PROGRAM p_Com_Modbus_RS485
VAR
	//Gestion de la com avec la passerelle LED
	Com_LED: Com485_Dalcnet;
	Lecture_Dimmer 	:INT;
	Lecture_Rouge 	:INT;
	Lecture_Vert 	:INT;
	Lecture_Bleu 	:INT;
	Lecture_Blanc 	:INT;
	LED_Com_Ok		:BOOL;
	LED_Com_Error	:BOOL;
	LED_Etape		:INT;
	
	//Gestion de la com avec GVL_RegTROX.Reg_Souf_GD_FCVT01
	FCVT01_Com_Ok		:BOOL;
	FCVT01_Com_Error	:BOOL;
	FCVT01_Etape		:INT;
	FCVT01_ConsAppli	:INT;
	
	//Gestion de la com avec GVL_RegTROX.Com_RegSouf_PD_FCVT02
	FCVT02_Com_Ok		:BOOL;
	FCVT02_Com_Error	:BOOL;
	FCVT02_Etape		:INT;
	FCVT02_ConsAppli	:INT;
	
	//Gestion de la com avec GVL_RegTROX.Com_RegSouf_Cabine_FCVT03
	FCVT03_Com_Ok		:BOOL;
	FCVT03_Com_Error	:BOOL;
	FCVT03_Etape		:INT;
	FCVT03_ConsAppli	:INT;
	
	//Gestion de la com avec GVL_RegTROX.Com_Reg_Bypass_FCVT04
	FCVT04_Com_Ok		:BOOL;
	FCVT04_Com_Error	:BOOL;
	FCVT04_Etape		:INT;
	FCVT04_ConsAppli	:INT;
	
	//Gestion de la com avec GVL_RegTROX.Com_RegSouf_CabGD_FCVT05
	FCVT05_Com_Ok		:BOOL;
	FCVT05_Com_Error	:BOOL;
	FCVT05_Etape		:INT;
	FCVT05_ConsAppli	:INT;
	
	//Gestion de la com avec GVL_RegTROX.Com_RegSouf_CabPD_FCVT06
	FCVT06_Com_Ok		:BOOL;
	FCVT06_Com_Error	:BOOL;
	FCVT06_Etape		:INT;
	FCVT06_ConsAppli	:INT;
	
	//Gestion de la com avec GVL_RegTROX.Com_RegRep_FCVT07
	FCVT07_Com_Ok		:BOOL;
	FCVT07_Com_Error	:BOOL;
	FCVT07_Etape		:INT;
	FCVT07_ConsAppli	:INT;
	
	Start_2: BOOL;
	Start_3: BOOL;
	Start_4: BOOL;
	Start_41: BOOL;
	Start_5: BOOL;
	Start_6: BOOL;
	Start_61: BOOL;
	Start_7: BOOL;
	Start_8: BOOL;
	Start_9: BOOL;
	FirstCycle: BOOL := TRUE;
	F_TRIG_0: F_TRIG;
	cpt: INT;
	CTU_Cpt: CTU;
	Cons_Cpt: WORD := 4;
	TOF_0: TOF;
	test: BOOL;
	
	//Gestion des forçages
	EF_FCVT01		:BOOL;
	F_FCVT01		:REAL;
	EF_FCVT02		:BOOL;
	F_FCVT02		:REAL;
	EF_FCVT03		:BOOL;
	F_FCVT03		:REAL;
	EF_FCVT04		:BOOL;
	F_FCVT04		:REAL;
	EF_FCVT05		:BOOL;
	F_FCVT05		:REAL;
	EF_FCVT06		:BOOL;
	F_FCVT06		:REAL;
	EF_FCVT07		:BOOL;
	F_FCVT07		:REAL;
END_VAR
VAR // added by the converter: edge detectors and wires of the graphical bodies
    _w1 : BOOL;
END_VAR

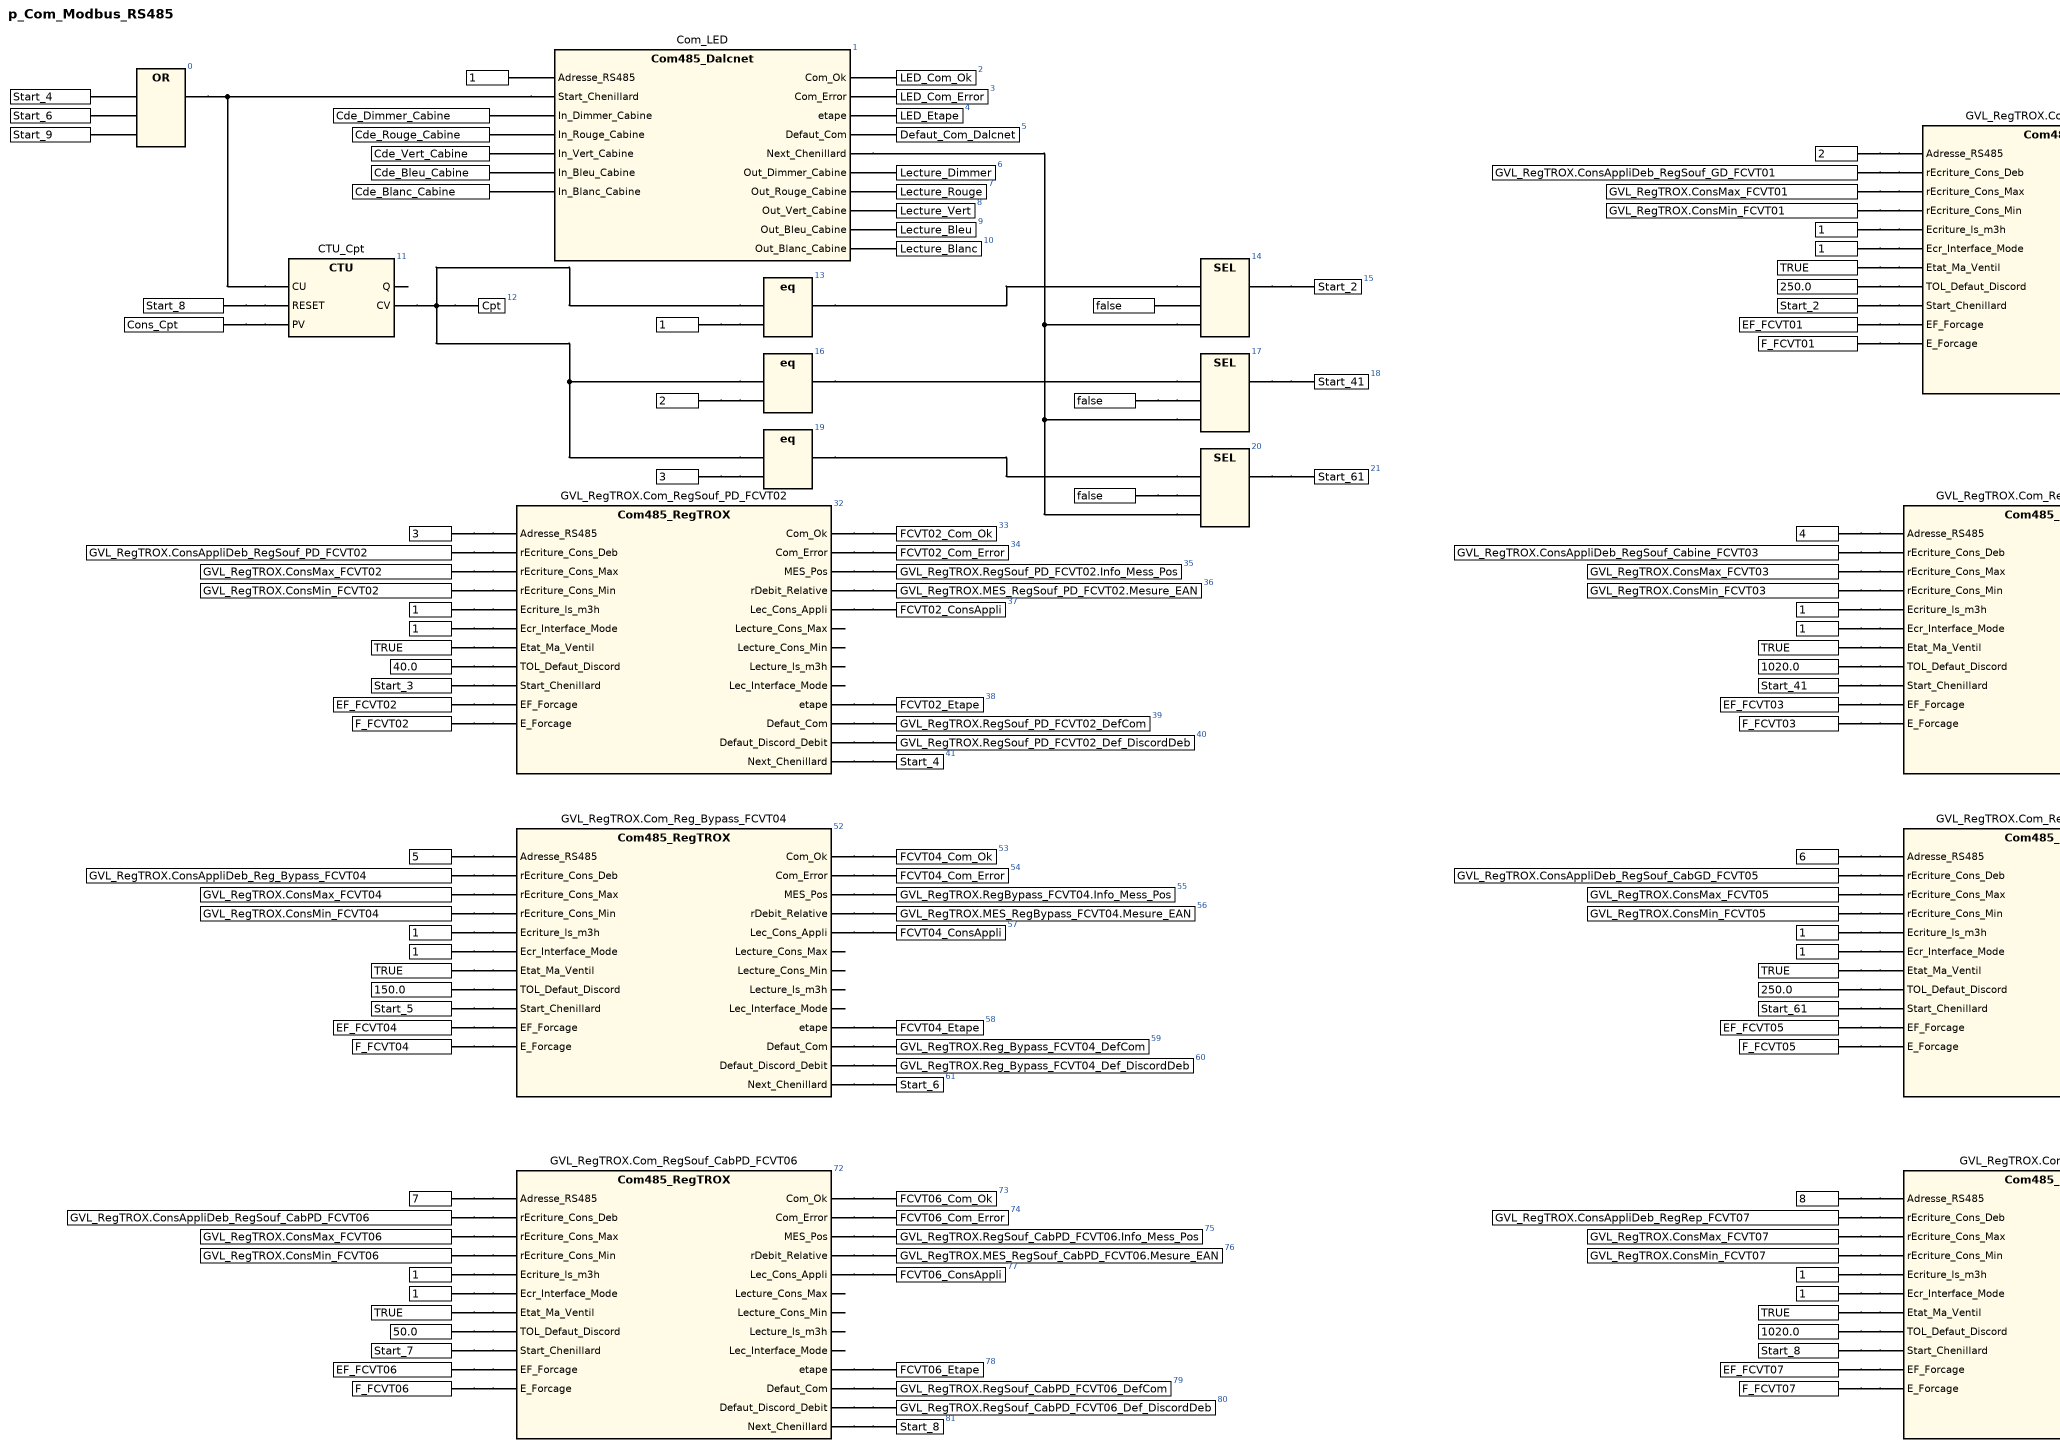
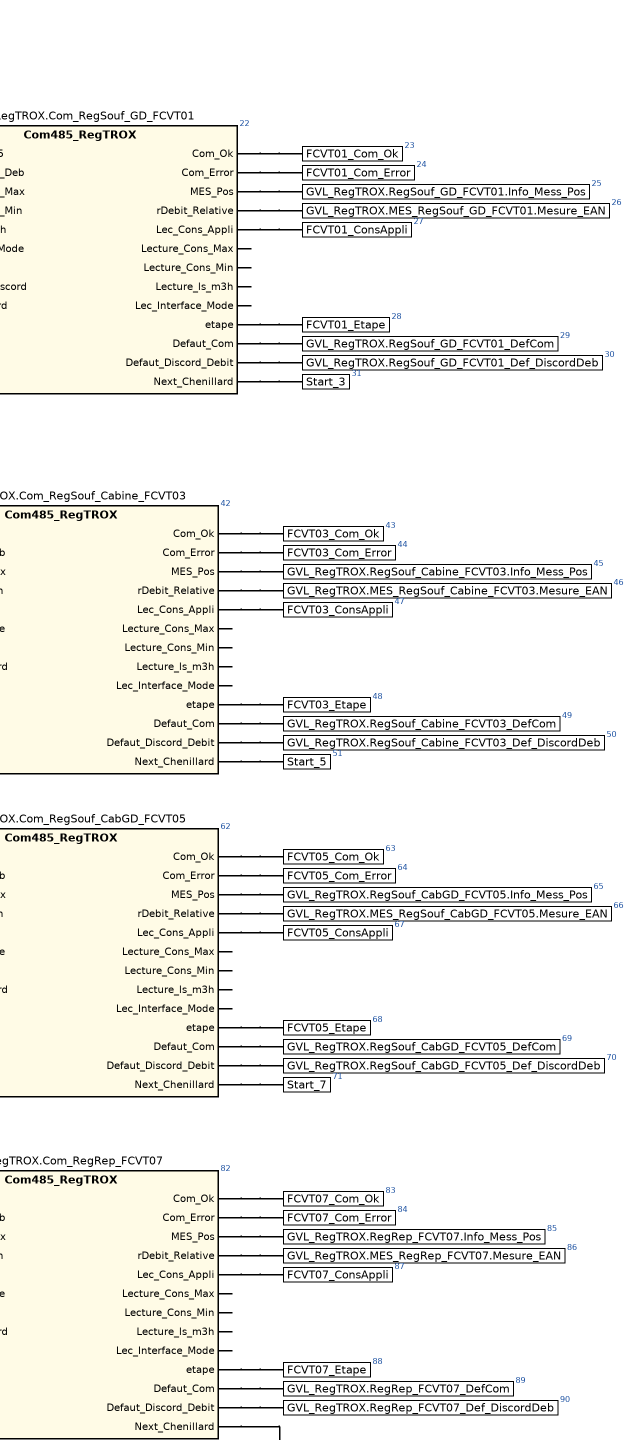
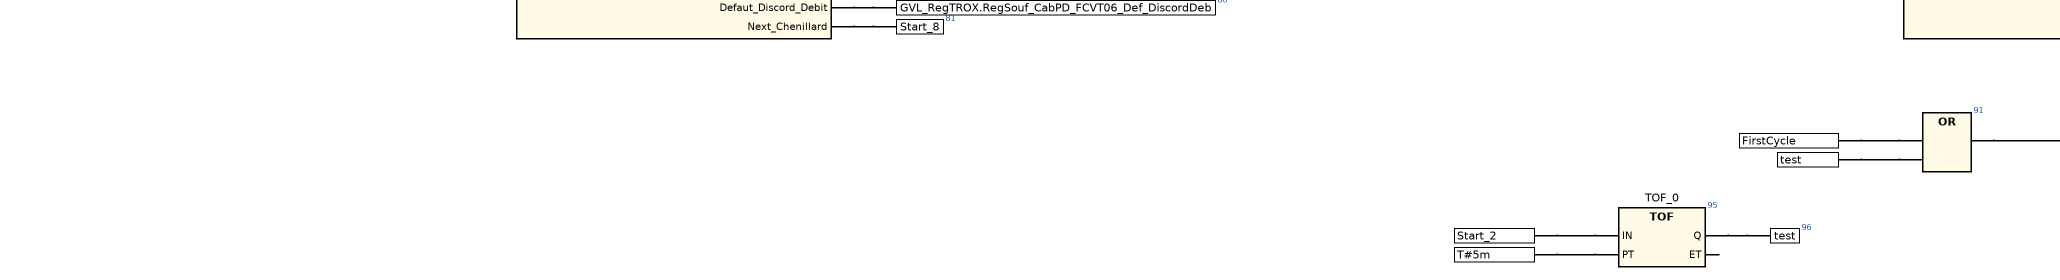
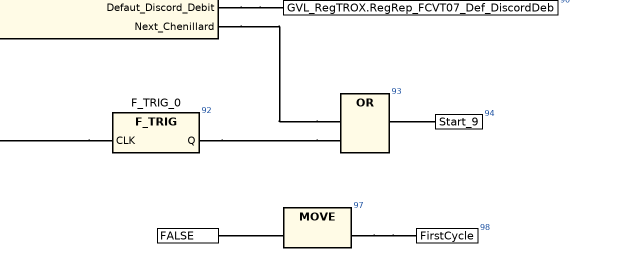
_w1 := Start_4 OR Start_6 OR Start_9;
Com_LED(
    Adresse_RS485 := 1,
    Start_Chenillard := _w1,
    In_Dimmer_Cabine := Cde_Dimmer_Cabine,
    In_Rouge_Cabine := Cde_Rouge_Cabine,
    In_Vert_Cabine := Cde_Vert_Cabine,
    In_Bleu_Cabine := Cde_Bleu_Cabine,
    In_Blanc_Cabine := Cde_Blanc_Cabine); // Com485_Dalcnet
LED_Com_Ok := Com_LED.Com_Ok;
LED_Com_Error := Com_LED.Com_Error;
LED_Etape := Com_LED.etape;
Defaut_Com_Dalcnet := Com_LED.Defaut_Com;
Lecture_Dimmer := Com_LED.Out_Dimmer_Cabine;
Lecture_Rouge := Com_LED.Out_Rouge_Cabine;
Lecture_Vert := Com_LED.Out_Vert_Cabine;
Lecture_Bleu := Com_LED.Out_Bleu_Cabine;
Lecture_Blanc := Com_LED.Out_Blanc_Cabine;
CTU_Cpt(CU := _w1, RESET := Start_8, PV := Cons_Cpt); // CTU
Cpt := CTU_Cpt.CV;
Start_2 := SEL(CTU_Cpt.CV = 1, false, Com_LED.Next_Chenillard);
Start_41 := SEL(CTU_Cpt.CV = 2, false, Com_LED.Next_Chenillard);
Start_61 := SEL(CTU_Cpt.CV = 3, false, Com_LED.Next_Chenillard);
GVL_RegTROX.Com_RegSouf_GD_FCVT01(
    Adresse_RS485 := 2,
    rEcriture_Cons_Deb := GVL_RegTROX.ConsAppliDeb_RegSouf_GD_FCVT01,
    rEcriture_Cons_Max := GVL_RegTROX.ConsMax_FCVT01,
    rEcriture_Cons_Min := GVL_RegTROX.ConsMin_FCVT01,
    Ecriture_ls_m3h := 1,
    Ecr_Interface_Mode := 1,
    Etat_Ma_Ventil := TRUE,
    TOL_Defaut_Discord := 250.0,
    Start_Chenillard := Start_2,
    EF_Forcage := EF_FCVT01,
    E_Forcage := F_FCVT01); // Com485_RegTROX
FCVT01_Com_Ok := GVL_RegTROX.Com_RegSouf_GD_FCVT01.Com_Ok;
FCVT01_Com_Error := GVL_RegTROX.Com_RegSouf_GD_FCVT01.Com_Error;
GVL_RegTROX.RegSouf_GD_FCVT01.Info_Mess_Pos := GVL_RegTROX.Com_RegSouf_GD_FCVT01.MES_Pos;
GVL_RegTROX.MES_RegSouf_GD_FCVT01.Mesure_EAN := GVL_RegTROX.Com_RegSouf_GD_FCVT01.rDebit_Relative;
FCVT01_ConsAppli := GVL_RegTROX.Com_RegSouf_GD_FCVT01.Lec_Cons_Appli;
FCVT01_Etape := GVL_RegTROX.Com_RegSouf_GD_FCVT01.etape;
GVL_RegTROX.RegSouf_GD_FCVT01_DefCom := GVL_RegTROX.Com_RegSouf_GD_FCVT01.Defaut_Com;
GVL_RegTROX.RegSouf_GD_FCVT01_Def_DiscordDeb := GVL_RegTROX.Com_RegSouf_GD_FCVT01.Defaut_Discord_Debit;
Start_3 := GVL_RegTROX.Com_RegSouf_GD_FCVT01.Next_Chenillard;
GVL_RegTROX.Com_RegSouf_PD_FCVT02(
    Adresse_RS485 := 3,
    rEcriture_Cons_Deb := GVL_RegTROX.ConsAppliDeb_RegSouf_PD_FCVT02,
    rEcriture_Cons_Max := GVL_RegTROX.ConsMax_FCVT02,
    rEcriture_Cons_Min := GVL_RegTROX.ConsMin_FCVT02,
    Ecriture_ls_m3h := 1,
    Ecr_Interface_Mode := 1,
    Etat_Ma_Ventil := TRUE,
    TOL_Defaut_Discord := 40.0,
    Start_Chenillard := Start_3,
    EF_Forcage := EF_FCVT02,
    E_Forcage := F_FCVT02); // Com485_RegTROX
FCVT02_Com_Ok := GVL_RegTROX.Com_RegSouf_PD_FCVT02.Com_Ok;
FCVT02_Com_Error := GVL_RegTROX.Com_RegSouf_PD_FCVT02.Com_Error;
GVL_RegTROX.RegSouf_PD_FCVT02.Info_Mess_Pos := GVL_RegTROX.Com_RegSouf_PD_FCVT02.MES_Pos;
GVL_RegTROX.MES_RegSouf_PD_FCVT02.Mesure_EAN := GVL_RegTROX.Com_RegSouf_PD_FCVT02.rDebit_Relative;
FCVT02_ConsAppli := GVL_RegTROX.Com_RegSouf_PD_FCVT02.Lec_Cons_Appli;
FCVT02_Etape := GVL_RegTROX.Com_RegSouf_PD_FCVT02.etape;
GVL_RegTROX.RegSouf_PD_FCVT02_DefCom := GVL_RegTROX.Com_RegSouf_PD_FCVT02.Defaut_Com;
GVL_RegTROX.RegSouf_PD_FCVT02_Def_DiscordDeb := GVL_RegTROX.Com_RegSouf_PD_FCVT02.Defaut_Discord_Debit;
Start_4 := GVL_RegTROX.Com_RegSouf_PD_FCVT02.Next_Chenillard;
GVL_RegTROX.Com_RegSouf_Cabine_FCVT03(
    Adresse_RS485 := 4,
    rEcriture_Cons_Deb := GVL_RegTROX.ConsAppliDeb_RegSouf_Cabine_FCVT03,
    rEcriture_Cons_Max := GVL_RegTROX.ConsMax_FCVT03,
    rEcriture_Cons_Min := GVL_RegTROX.ConsMin_FCVT03,
    Ecriture_ls_m3h := 1,
    Ecr_Interface_Mode := 1,
    Etat_Ma_Ventil := TRUE,
    TOL_Defaut_Discord := 1020.0,
    Start_Chenillard := Start_41,
    EF_Forcage := EF_FCVT03,
    E_Forcage := F_FCVT03); // Com485_RegTROX
FCVT03_Com_Ok := GVL_RegTROX.Com_RegSouf_Cabine_FCVT03.Com_Ok;
FCVT03_Com_Error := GVL_RegTROX.Com_RegSouf_Cabine_FCVT03.Com_Error;
GVL_RegTROX.RegSouf_Cabine_FCVT03.Info_Mess_Pos := GVL_RegTROX.Com_RegSouf_Cabine_FCVT03.MES_Pos;
GVL_RegTROX.MES_RegSouf_Cabine_FCVT03.Mesure_EAN := GVL_RegTROX.Com_RegSouf_Cabine_FCVT03.rDebit_Relative;
FCVT03_ConsAppli := GVL_RegTROX.Com_RegSouf_Cabine_FCVT03.Lec_Cons_Appli;
FCVT03_Etape := GVL_RegTROX.Com_RegSouf_Cabine_FCVT03.etape;
GVL_RegTROX.RegSouf_Cabine_FCVT03_DefCom := GVL_RegTROX.Com_RegSouf_Cabine_FCVT03.Defaut_Com;
GVL_RegTROX.RegSouf_Cabine_FCVT03_Def_DiscordDeb := GVL_RegTROX.Com_RegSouf_Cabine_FCVT03.Defaut_Discord_Debit;
Start_5 := GVL_RegTROX.Com_RegSouf_Cabine_FCVT03.Next_Chenillard;
GVL_RegTROX.Com_Reg_Bypass_FCVT04(
    Adresse_RS485 := 5,
    rEcriture_Cons_Deb := GVL_RegTROX.ConsAppliDeb_Reg_Bypass_FCVT04,
    rEcriture_Cons_Max := GVL_RegTROX.ConsMax_FCVT04,
    rEcriture_Cons_Min := GVL_RegTROX.ConsMin_FCVT04,
    Ecriture_ls_m3h := 1,
    Ecr_Interface_Mode := 1,
    Etat_Ma_Ventil := TRUE,
    TOL_Defaut_Discord := 150.0,
    Start_Chenillard := Start_5,
    EF_Forcage := EF_FCVT04,
    E_Forcage := F_FCVT04); // Com485_RegTROX
FCVT04_Com_Ok := GVL_RegTROX.Com_Reg_Bypass_FCVT04.Com_Ok;
FCVT04_Com_Error := GVL_RegTROX.Com_Reg_Bypass_FCVT04.Com_Error;
GVL_RegTROX.RegBypass_FCVT04.Info_Mess_Pos := GVL_RegTROX.Com_Reg_Bypass_FCVT04.MES_Pos;
GVL_RegTROX.MES_RegBypass_FCVT04.Mesure_EAN := GVL_RegTROX.Com_Reg_Bypass_FCVT04.rDebit_Relative;
FCVT04_ConsAppli := GVL_RegTROX.Com_Reg_Bypass_FCVT04.Lec_Cons_Appli;
FCVT04_Etape := GVL_RegTROX.Com_Reg_Bypass_FCVT04.etape;
GVL_RegTROX.Reg_Bypass_FCVT04_DefCom := GVL_RegTROX.Com_Reg_Bypass_FCVT04.Defaut_Com;
GVL_RegTROX.Reg_Bypass_FCVT04_Def_DiscordDeb := GVL_RegTROX.Com_Reg_Bypass_FCVT04.Defaut_Discord_Debit;
Start_6 := GVL_RegTROX.Com_Reg_Bypass_FCVT04.Next_Chenillard;
GVL_RegTROX.Com_RegSouf_CabGD_FCVT05(
    Adresse_RS485 := 6,
    rEcriture_Cons_Deb := GVL_RegTROX.ConsAppliDeb_RegSouf_CabGD_FCVT05,
    rEcriture_Cons_Max := GVL_RegTROX.ConsMax_FCVT05,
    rEcriture_Cons_Min := GVL_RegTROX.ConsMin_FCVT05,
    Ecriture_ls_m3h := 1,
    Ecr_Interface_Mode := 1,
    Etat_Ma_Ventil := TRUE,
    TOL_Defaut_Discord := 250.0,
    Start_Chenillard := Start_61,
    EF_Forcage := EF_FCVT05,
    E_Forcage := F_FCVT05); // Com485_RegTROX
FCVT05_Com_Ok := GVL_RegTROX.Com_RegSouf_CabGD_FCVT05.Com_Ok;
FCVT05_Com_Error := GVL_RegTROX.Com_RegSouf_CabGD_FCVT05.Com_Error;
GVL_RegTROX.RegSouf_CabGD_FCVT05.Info_Mess_Pos := GVL_RegTROX.Com_RegSouf_CabGD_FCVT05.MES_Pos;
GVL_RegTROX.MES_RegSouf_CabGD_FCVT05.Mesure_EAN := GVL_RegTROX.Com_RegSouf_CabGD_FCVT05.rDebit_Relative;
FCVT05_ConsAppli := GVL_RegTROX.Com_RegSouf_CabGD_FCVT05.Lec_Cons_Appli;
FCVT05_Etape := GVL_RegTROX.Com_RegSouf_CabGD_FCVT05.etape;
GVL_RegTROX.RegSouf_CabGD_FCVT05_DefCom := GVL_RegTROX.Com_RegSouf_CabGD_FCVT05.Defaut_Com;
GVL_RegTROX.RegSouf_CabGD_FCVT05_Def_DiscordDeb := GVL_RegTROX.Com_RegSouf_CabGD_FCVT05.Defaut_Discord_Debit;
Start_7 := GVL_RegTROX.Com_RegSouf_CabGD_FCVT05.Next_Chenillard;
GVL_RegTROX.Com_RegSouf_CabPD_FCVT06(
    Adresse_RS485 := 7,
    rEcriture_Cons_Deb := GVL_RegTROX.ConsAppliDeb_RegSouf_CabPD_FCVT06,
    rEcriture_Cons_Max := GVL_RegTROX.ConsMax_FCVT06,
    rEcriture_Cons_Min := GVL_RegTROX.ConsMin_FCVT06,
    Ecriture_ls_m3h := 1,
    Ecr_Interface_Mode := 1,
    Etat_Ma_Ventil := TRUE,
    TOL_Defaut_Discord := 50.0,
    Start_Chenillard := Start_7,
    EF_Forcage := EF_FCVT06,
    E_Forcage := F_FCVT06); // Com485_RegTROX
FCVT06_Com_Ok := GVL_RegTROX.Com_RegSouf_CabPD_FCVT06.Com_Ok;
FCVT06_Com_Error := GVL_RegTROX.Com_RegSouf_CabPD_FCVT06.Com_Error;
GVL_RegTROX.RegSouf_CabPD_FCVT06.Info_Mess_Pos := GVL_RegTROX.Com_RegSouf_CabPD_FCVT06.MES_Pos;
GVL_RegTROX.MES_RegSouf_CabPD_FCVT06.Mesure_EAN := GVL_RegTROX.Com_RegSouf_CabPD_FCVT06.rDebit_Relative;
FCVT06_ConsAppli := GVL_RegTROX.Com_RegSouf_CabPD_FCVT06.Lec_Cons_Appli;
FCVT06_Etape := GVL_RegTROX.Com_RegSouf_CabPD_FCVT06.etape;
GVL_RegTROX.RegSouf_CabPD_FCVT06_DefCom := GVL_RegTROX.Com_RegSouf_CabPD_FCVT06.Defaut_Com;
GVL_RegTROX.RegSouf_CabPD_FCVT06_Def_DiscordDeb := GVL_RegTROX.Com_RegSouf_CabPD_FCVT06.Defaut_Discord_Debit;
Start_8 := GVL_RegTROX.Com_RegSouf_CabPD_FCVT06.Next_Chenillard;
GVL_RegTROX.Com_RegRep_FCVT07(
    Adresse_RS485 := 8,
    rEcriture_Cons_Deb := GVL_RegTROX.ConsAppliDeb_RegRep_FCVT07,
    rEcriture_Cons_Max := GVL_RegTROX.ConsMax_FCVT07,
    rEcriture_Cons_Min := GVL_RegTROX.ConsMin_FCVT07,
    Ecriture_ls_m3h := 1,
    Ecr_Interface_Mode := 1,
    Etat_Ma_Ventil := TRUE,
    TOL_Defaut_Discord := 1020.0,
    Start_Chenillard := Start_8,
    EF_Forcage := EF_FCVT07,
    E_Forcage := F_FCVT07); // Com485_RegTROX
FCVT07_Com_Ok := GVL_RegTROX.Com_RegRep_FCVT07.Com_Ok;
FCVT07_Com_Error := GVL_RegTROX.Com_RegRep_FCVT07.Com_Error;
GVL_RegTROX.RegRep_FCVT07.Info_Mess_Pos := GVL_RegTROX.Com_RegRep_FCVT07.MES_Pos;
GVL_RegTROX.MES_RegRep_FCVT07.Mesure_EAN := GVL_RegTROX.Com_RegRep_FCVT07.rDebit_Relative;
FCVT07_ConsAppli := GVL_RegTROX.Com_RegRep_FCVT07.Lec_Cons_Appli;
FCVT07_Etape := GVL_RegTROX.Com_RegRep_FCVT07.etape;
GVL_RegTROX.RegRep_FCVT07_DefCom := GVL_RegTROX.Com_RegRep_FCVT07.Defaut_Com;
GVL_RegTROX.RegRep_FCVT07_Def_DiscordDeb := GVL_RegTROX.Com_RegRep_FCVT07.Defaut_Discord_Debit;
F_TRIG_0(CLK := FirstCycle OR test); // F_TRIG
Start_9 := GVL_RegTROX.Com_RegRep_FCVT07.Next_Chenillard OR F_TRIG_0.Q;
TOF_0(IN := Start_2, PT := T#5m); // TOF
test := TOF_0.Q;
FirstCycle := FALSE;

END_PROGRAM

(* stored: Version 1.1.0.1, ProductVersion 3.1.4024.16
   POU p_Com_Modbus_RS485: Id {8e5554ef-f93f-4641-b8b8-3aece345f156}, SpecialFunc None *)
